FUNCTION_BLOCK ActiveLogic
VAR_INPUT
END_VAR
VAR_OUTPUT
END_VAR
VAR
END_VAR

LocalVariables.Locations[1].Active := gvl.PistonInputForward;
LocalVariables.Locations[2].Active := gvl.MotorTableMove;
LocalVariables.Locations[3].Active := gvl.PistonPress;
LocalVariables.Locations[4].Active := gvl.PistonOutputForward;
LocalVariables.Locations[5].Active := gvl.MotorBeltMove;
LocalVariables.Locations[6].Active := NOT gvl.FotocellOutput;

END_FUNCTION_BLOCK

(* stored: Version 1.1.0.1, ProductVersion 3.1.4024.12
   POU ActiveLogic: Id {a18fb611-4c29-4205-b06a-1f2633a95e85}, SpecialFunc None *)
